(*
SPDX-FileCopyrightText: © 2026 Oleksandr Tiutyk <trofimich@gmail.com>
SPDX-License-Identifier: MIT
License: https://opensource.org/license/mit
*)

INTERFACE IDataMemberTypeClassNotSupportedException EXTENDS IGeneralException

METHOD Throw
VAR_INPUT
	sourceNamespaceName : STRING;
	sourceClassName : STRING;
	sourcePOUName : STRING;
	sourcePosition : STRING;
	dataMemberName : STRING;
	dataMemberType : __SYSTEM.TYPE_CLASS;
END_VAR
END_METHOD

END_INTERFACE

(* stored: Version 1.1.0.1
   Itf IDataMemberTypeClassNotSupportedException: Id {a45d046e-cfd6-46af-9060-568a379f671e}
   Method Throw: Id {5803b728-3de8-4545-8f65-0e2db12e9b94} *)
